Staubli VAL3: JointForce.dtx

public num jf1
public num jf2
public num jf3
public num jf4
public num jf5
public num jf6
